FUNCTION_BLOCK Fb_Test
VAR_INPUT
END_VAR
VAR_OUTPUT
END_VAR
VAR
END_VAR

END_FUNCTION_BLOCK

(* stored: Version 1.1.0.1, ProductVersion 3.1.4024.12
   POU Fb_Test: Id {d3d0c43f-c219-45f2-ba4d-2a7f41afbcfe}, SpecialFunc None *)
